(* IEC 61131-3 sources: mect_apps/TP1043_01_A/Wattmeter_PLC, 3 files *)

(* ---- Resource1.gvl ---- *)
(* Global variable file *)
VAR_GLOBAL

END_VAR

(* ---- Init.st ---- *)
(*[[
]]*)
PROGRAM Init
#import "Crosstable.gvl"
#import "Resource1.gvl"
VAR
END_VAR

	PLC_timeWin := 60.0;

END_PROGRAM

(* ---- Slow.st ---- *)
(*[[
]]*)
PROGRAM Slow
#import "Crosstable.gvl"
#import "Resource1.gvl"
VAR
END_VAR

;
END_PROGRAM
